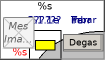
VISUALIZATION VISU_JAUGE_BCG450_V_HAUT_ETHERCAT  // 105x60
VAR_IN_OUT
	m_Input_JAUGE : BLOCK_BCG450_ETHERCAT;
END_VAR
    Rectangle (0,0 105x60), invisible if: TRUE
    Rectangle (0,10 90x20), "??????", invisible if: (m_Input_JAUGE.STATE_OK) <> 0
    Group (31,31 28x28)
        Ellipse (0,0 140x100)
        Rectangle (0,50 140x150)
        Polyline (140,50)
    Rectangle (35,40 20x10), colour toggle: NOT ( m_Input_JAUGE.OP_RAH.Etape.4 OR m_Input_JAUGE.OP_RAH.Etape.5 OR m_Input_JAUGE.OP_RAH.Etape.6 OR m_Input_JAUGE.OP_RAH.Etape.7), invisible if: (m_Input_JAUGE.OP_DGZ.EC) <> 0
    Rectangle (10,1 70x10), "%s", text variable: m_Input_JAUGE.MNEMO
    Rectangle (35,40 20x10), invisible if: NOT m_Input_JAUGE.OP_DGZ.EC
    Rectangle (29,30 32x30), invisible if: NOT (m_Input_JAUGE.Autor_ON_IHM OR m_Input_JAUGE.Autor_Off_IHM ) OR NOT PRG_User.ACTU_USER.MAINTENANCE
        tap m_Input_JAUGE.M_M1
    Group (5,10 88x18), invisible if: NOT m_Input_JAUGE.STATE_OK
        Rectangle (0,0 57x20), "%1.1e", text variable: m_Input_JAUGE.STATE_Pression
        Rectangle (60,0 27x20), "Torr", invisible if: NOT (m_Input_JAUGE.CONF_unit = 1)
        Rectangle (60,0 30x20), "mbar", invisible if: NOT (m_Input_JAUGE.CONF_unit = 0)
        Rectangle (60,0 27x20), "Pa", invisible if: NOT (m_Input_JAUGE.CONF_unit = 2)
    Rectangle (5,47 30x10), "%s", text variable: m_Input_JAUGE.STATE_ERR, invisible if: NOT m_Input_JAUGE.STATE_NOK
    Image (3,17 31x31), invisible if: NOT m_Input_JAUGE.STATE_NOK, image: MesImages.warning
    Button (63,34 40x17), "Degas", invisible if: NOT m_Input_JAUGE.AUTOR_Dgz_IHM OR NOT PRG_User.ACTU_USER.MAINTENANCE
        toggle m_Input_JAUGE.M_DGZ
END_VISUALIZATION

(* stored: Version 1.1.0.1, ProductVersion 3.1.4024.10
   Visu VISU_JAUGE_BCG450_V_HAUT_ETHERCAT: Id {cf32ca16-dc70-4ec9-9717-d3f6b18b5866} *)
